ABB RobotStudio station: save_station.rsstn

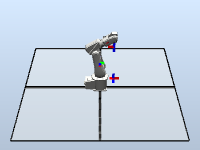
Station Station (saved by RobotStudio 6.7.7936.1011)
Controller WILL4230
  mechanical unit ROB_1: IRB120_3_58__01, 6 joints, base frame (0, 0, 0) mm
Layout (positions relative to the parent item):
  - IRB120_3_58__01 [mechanism, from Robots\IRB120_3_58_G_01.rslib] at (0, 0, 0) mm; joint values [0, -0.1947, -0.3256, 0, 2.0911, 0] (rad or m)
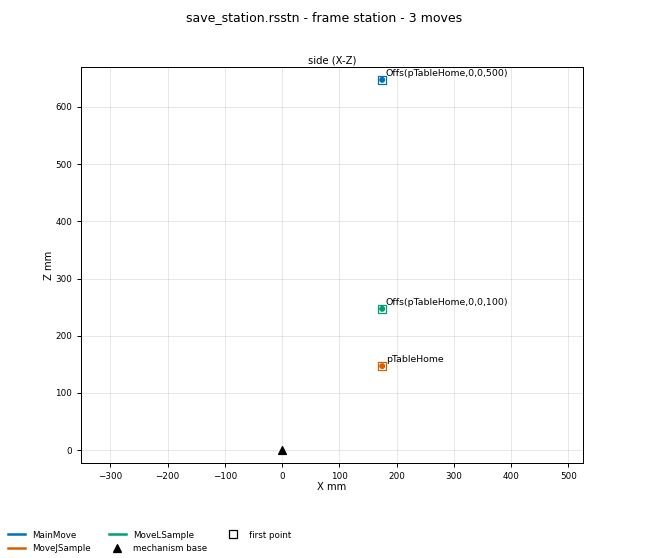
[picture p0: tool path of save_station.rsstn in frame station, 3 of 7 moves have a stored position in this frame; points joined in program order, loops and branches not executed]
Targets, tools, work objects and paths stored in the station, written as RAPID:
! task T_ROB1
MODULE MTRN_Rob_Data
  PERS tooldata tSCup:=[TRUE,[[0,0,65],[1,0,0,0]],[0.5,[0,0,20],[1,0,0,0],0,0,0]];
  PERS wobjdata wTable:=[FALSE,TRUE,"",[[175,0,147],[1,0,0,0]],[[0,0,0],[1,0,0,0]]];
  PERS wobjdata wConv:=[FALSE,TRUE,"",[[50,184,22],[0.5,-0.5,0.5,0.5]],[[1,1,1],[1,0,0,0]]];
  CONST robtarget pTableHome:=[[175,0,147],[0,0,-1,0],[0,0,0,0],[9E+09,9E+09,9E+09,9E+09,9E+09,9E+09]];
  CONST jointtarget jtCalibPos:=[[-90,0,0,0,0,0],[9E+09,9E+09,9E+09,9E+09,9E+09,9E+09]];
ENDMODULE

! task T_ROB1
MODULE MTRN4230_Server_Sample
  PROC CloseConnection()
  ENDPROC
  PROC MainServer()
    ListenForAndAcceptConnection;
    CloseConnection;
  ENDPROC
  PROC Main1()
    MainServer;
  ENDPROC
  PROC ListenForAndAcceptConnection()
  ENDPROC
ENDMODULE

! task T_ROB1
MODULE MTRN4230_Move_Sample
  PROC MainMove()
    MoveToCalibPos;
    MoveJSample;
    MoveLSample;
    MoveL Offs(pTableHome, 0, 0, 500),v100,fine,tSCup;
  ENDPROC
  PROC MoveJSample()
    MoveJ pTableHome,v100,fine,tSCup;
  ENDPROC
  PROC MoveLSample()
    MoveL Offs(pTableHome, 0, 0, 100),v100,fine,tSCup;
  ENDPROC
ENDMODULE

! task T_ROB1
MODULE MTRN4230_IO_Sample
  PROC Main()
    MainIO;
  ENDPROC
  PROC MainIO()
    TurnVacOn;
    WaitTime 2;
    TurnVacOff;
    TurnConOnSafely;
    WaitTime 2;
    TurnConOff;
  ENDPROC
  PROC TurnVacOn()
    SetDO DO10_1,1;
  ENDPROC
  PROC TurnVacOff()
    SetDO DO10_1,0;
  ENDPROC
  PROC TurnConOnSafely()
    SetDO DO10_3,1;
    SetDO DO10_3,0;
  ENDPROC
  PROC TurnConOff()
    SetDO DO10_3,0;
  ENDPROC
ENDMODULE

! task T_ROB1
MODULE MTRN_Rob_Proc
  PROC MoveToCalibPos()
    MoveAbsJ jtCalibPos,v400,fine,tool0;
  ENDPROC
ENDMODULE

! task T_ROB1
MODULE Assignment2
  PROC MainAss2()
    MoveToCalibPos;
    vacPwrOn;
    vacSolOn;
    MoveL Offs(testTarget, 0, 0, 500),v100,fine,tScup;
    MoveL Offs(testTarget, 0, 100, 500),v100,fine,tSCup;
    MoveL Offs(testTarget, 0, 100, 5),v100,fine,tSCup;
    vacSolOff;
    vacPwerOff;
    MoveToCalibPos;
  ENDPROC
  PROC vacPwrOn()
    SetDO DO10_1,1;
  ENDPROC
  PROC vacPwerOff()
    SetDO DO10_1,0;
  ENDPROC
  PROC vacSolOn()
    SetDO DO10_2,1;
  ENDPROC
  PROC vacSolOff()
    SetDO DO10_2,0;
  ENDPROC
  PROC conRunOn()
    SetDO DO10_3,1;
  ENDPROC
  PROC conRunOff()
    SetDO DO10_3,0;
  ENDPROC
  PROC conDirRob()
    SetDO DO10_4,1;
  ENDPROC
  PROC conDirHome()
    SetDO DO10_4,0;
  ENDPROC
ENDMODULE

